Staubli VAL3: Welcome.pjx

--- Welcome.pjx ---
Parameters version=s7.9 stackSize=5000 millimeterUnit=true
Program file=start.pgx
Program file=stop.pgx
Data file=Welcome.dtx

--- Welcome.dtx ---
mdesc mNomSpeed

--- start.pgx ---
program start()
begin
  while true
    delay(0)
  endWhile
end
